PROGRAM MAIN
VAR
END_VAR

PG_Time();
PG_Alarm();
PG_Calculate_Sun();
PG_Rain();
PG_Heizung();
PG_Wind();
PG_Visu();
PG_Besucher();
PG_SimulationsHaus();

END_PROGRAM

(* stored: Version 1.1.0.1, ProductVersion 3.1.4018.5
   POU MAIN: Id {b35740f0-740b-4f7e-bcd7-59db9c475d00}, SpecialFunc None *)
